FUNCTION_BLOCK RoomInterface IMPLEMENTS I_Room
VAR_STAT
	_nMaxRoom	: UDINT;
END_VAR

VAR
	_ctx		: REFERENCE TO Room_Ctx;
	_nId		: UDINT;
END_VAR

//FB_Init is always available implicitly and it is used primarily for initialization.
//The return value is not evaluated. For a specific influence, you can also declare the
//methods explicitly and provide additional code there with the standard initialization
//code. You can evaluate the return value.
METHOD FB_Init: BOOL
VAR_INPUT
    bInitRetains: BOOL; // TRUE: the retain variables are initialized (reset warm / reset cold)
    bInCopyCode: BOOL;  // TRUE: the instance will be copied to the copy code afterward (online change)
	
	ctx			: REFERENCE TO Room_Ctx;
END_VAR
_ctx REF= ctx;
_ctx.priv.iThisRoom := THIS^;
_nMaxRoom := _nMaxRoom + 1;
_nId := _nMaxRoom;
_ctx.hmi.nId := _nMaxRoom;
END_METHOD

METHOD GoIdle
IF NOT _ctx.priv.bActive THEN
	RETURN;
END_IF

_ctx.state.iMgr.Request(_ctx.state.iIdle);
END_METHOD

PROPERTY Id : UDINT
GET
Id := _nId;
END_GET
END_PROPERTY

PROPERTY IsActive : BOOL
GET
IsActive := _ctx.priv.bActive;
END_GET
END_PROPERTY

PROPERTY IsClosed : BOOL
GET
IsClosed := _ctx.priv.bClosed;
END_GET
END_PROPERTY

PROPERTY IsOpen : BOOL
GET
IsOpen := _ctx.priv.bOpen;
END_GET
END_PROPERTY

PROPERTY IsReady : BOOL
GET
IsReady := _ctx.priv.bReady;
END_GET
END_PROPERTY

METHOD Open
IF NOT _ctx.priv.bActive THEN
	RETURN;
END_IF

_ctx.io.bOpenValves := TRUE;
END_METHOD

PROPERTY Timeout : TIME
GET
Timeout := UDINT_TO_TIME(_ctx.hmi.nTimeout * 1000 * 60);
END_GET
END_PROPERTY

METHOD TriggerFault
VAR_INPUT
	sErrorText		: Str;
END_VAR
_ctx.hmi.sErrorText := sErrorText;
_ctx.state.iMgr.Request(_ctx.state.iFault);
END_METHOD

END_FUNCTION_BLOCK

(* stored: Version 1.1.0.1
   POU RoomInterface: Id {6599786c-ba93-4fed-b30a-839e05cc02d4}, SpecialFunc None
   Method FB_init: Id {ca22bbab-be21-4373-9409-1f9b1007feee}
   Method GoIdle: Id {a7b9d657-00fa-45e9-baeb-af69e6018523}
   Property Id: Id {cab61793-e91a-43d3-b4f1-43fa7063eb1d}
   Get Get: Id {0db4bec7-83f4-40cb-a9f0-f42887b91727}
   Property IsActive: Id {05099b11-7bf8-4c59-9cb6-a7bb7b3a2db4}
   Get Get: Id {9fda7680-eecb-4790-855c-e58914c1503a}
   Property IsClosed: Id {8201ff4f-9b53-446e-b50e-9f3ccbca46fc}
   Get Get: Id {860a5c51-d17a-487c-8cbf-c0e50bf3bb19}
   Property IsOpen: Id {363ee4e3-517b-4e8e-a8ef-3e40d440e3f6}
   Get Get: Id {19a270b5-a546-429e-9caa-5fce82d24831}
   Property IsReady: Id {faede1ff-4852-4edb-be53-dba65663064d}
   Get Get: Id {9ff15937-25cb-474e-b7f4-31a6db2c8096}
   Method Open: Id {2ef519f7-2d21-4fe3-a50b-7c53dc7ef0e6}
   Property Timeout: Id {eecc649b-322a-4026-a5ac-c0aea4a056f0}
   Get Get: Id {2bf87570-2da5-4e3e-8bee-0d0856799639}
   Method TriggerFault: Id {58bcbc1a-fac3-413a-a2a2-69cf90b35fc2} *)
